PROGRAM P_Visu
VAR
	bFirstRun					: BOOL := TRUE;	
	
END_VAR

IF bFirstRun THEN
	bFirstRun := FALSE;
	FirstRun();
END_IF

JogButton();
SwitchButton();
SyncVariable();

METHOD FirstRun : BOOL
VAR_INPUT
END_VAR
GVL_VISU.stMachineConfig := P_Machine.MachineConfig;	
GVL_VISU.stCurMat := fbmat.Mat;
END_METHOD

METHOD JogButton : BOOL
VAR_INPUT
END_VAR
// JOG X
IF GVL_VISU.stMaintCmds.bJogXBw THEN
	GVL.fbMatAndToolHandling.JogX(TRUE);
ELSIF GVL_VISU.stMaintCmds.bJogXFw THEN
	GVL.fbMatAndToolHandling.JogX(FALSE);
ELSE
	GVL.fbMatAndToolHandling.JogXStop();
END_IF

// JOG Y
IF GVL_VISU.stMaintCmds.bJogYBw THEN
	GVL.fbMatAndToolHandling.JogY(TRUE);
ELSIF GVL_VISU.stMaintCmds.bJogYFw THEN
	GVL.fbMatAndToolHandling.JogY(FALSE);
ELSE
	GVL.fbMatAndToolHandling.JogYStop();
END_IF

// JOG Punch
IF GVL_VISU.stMaintCmds.bJogPunchBw THEN
	GVL.fbPunchEngine.Jog(FALSE, TRUE);
ELSIF GVL_VISU.stMaintCmds.bJogPunchFw THEN
	GVL.fbPunchEngine.Jog(TRUE, FALSE);
ELSE
	GVL.fbPunchEngine.JogStop();
END_IF

// JOG BELT
IF GVL_VISU.stMaintCmds.bJogOutletBelt THEN
	GVL.fbPunchEngine.OutletBeltJog(TRUE);
ELSE
	GVL.fbPunchEngine.OutletBeltJog(FALSE);
END_IF
END_METHOD

METHOD SwitchButton : BOOL
VAR_STAT
	stNullPunchCmds				: ST_PunchCmds;
	stNullMaintCmds				: ST_MaintCmds;
END_VAR
// PUNCH COMMANDS
IF MEMCMP(ADR(GVL_VISU.stPunchCmds), ADR(stNullPunchCmds), SIZEOF(ST_PunchCmds)) <> 0 THEN
	IF GVL_VISU.stPunchCmds.bLoad THEN
		P_Machine.LoadMat(GVL_VISU.stCurMat);		
		P_Machine.LoadJob(GVL_VISU.stPunchJob);	
	END_IF
	
	IF GVL_VISU.stPunchCmds.bStart THEN	
		P_Machine.LoadMat(GVL_VISU.stCurMat);	
		P_Machine.Start(GVL_VISU.stPunchJob);	
	END_IF
	
	IF GVL_VISU.stPunchCmds.bStop THEN
		P_Machine.Stop();	
	END_IF
	
	IF GVL_VISU.stPunchCmds.bResume THEN
		P_Machine.Resume();	
	END_IF
	
	IF GVL_VISU.stPunchCmds.bHalt THEN
		P_Machine.ClearJob();
		P_Machine.Halt();	
	END_IF	
		
	IF GVL_VISU.stPunchCmds.bLoadLeft THEN
		P_Machine.Maint(TRUE, TRUE, FALSE);	
	END_IF	
	
	IF GVL_VISU.stPunchCmds.bLoadRight THEN
		P_Machine.Maint(TRUE, TRUE, TRUE);	
	END_IF	
	
	IF GVL_VISU.stPunchCmds.bLoadStop THEN
		P_Machine.Halt();	
	END_IF	
	
	IF GVL_VISU.stPunchCmds.bUnlock THEN
		IF fbSafetyLock.Locked THEN
			GVL.fbSafetyLock.Unlock();
		ELSE
			GVL.fbSafetyLock.Lock();
		END_IF
	END_IF		
	
	IF GVL_VISU.stPunchCmds.bMoveTDC THEN
		GVL.fbPunchEngine.MoveTDC();	
	END_IF	
	
	IF GVL_VISU.stPunchCmds.bOutletBelt THEN
		GVL.fbPunchEngine.OutletBeltOnce();	
	END_IF	
		
	IF GVL_VISU.stPunchCmds.bOverride THEN
		P_Machine.Override := GVL_VISU.stPunchParam.fOverride;
	END_IF	
END_IF

// RESET PUNCH COMMANDS
GVL_VISU.stPunchCmds.bLoad := FALSE;
GVL_VISU.stPunchCmds.bStart := FALSE;
GVL_VISU.stPunchCmds.bStop := FALSE;
GVL_VISU.stPunchCmds.bResume := FALSE;
GVL_VISU.stPunchCmds.bHalt := FALSE;
GVL_VISU.stPunchCmds.bLoadLeft := FALSE;
GVL_VISU.stPunchCmds.bLoadRight := FALSE;
GVL_VISU.stPunchCmds.bMoveTDC := FALSE;
GVL_VISU.stPunchCmds.bOutletBelt := FALSE;
GVL_VISU.stPunchCmds.bOverride := FALSE;
GVL_VISU.stPunchCmds.bUnlock := FALSE;
GVL_VISU.stPunchCmds.bLoadStop := FALSE;

// MAINT COMMANDS
IF MEMCMP(ADR(GVL_VISU.stMaintCmds), ADR(stNullMaintCmds), SIZEOF(ST_MaintCmds)) <> 0 THEN	
	IF GVL_VISU.stMaintCmds.bLoadConfig THEN
		P_Machine.LoadConfig(GVL_VISU.stMachineConfig);
	END_IF
	
	IF GVL_VISU.stMaintCmds.bChangeTool THEN
		GVL.fbMatAndToolHandling.ChangeTool(GVL_VISU.stMaintParam.nChangeTool);
	END_IF
	
	IF GVL_VISU.stMaintCmds.bMoveXYMaint THEN
		P_Machine.Maint(TRUE, TRUE, FALSE);	
	END_IF
	
	IF GVL_VISU.stMaintCmds.bMoveXYMaintAlt THEN
		P_Machine.Maint(TRUE, TRUE, TRUE);	
	END_IF
	
	IF GVL_VISU.stMaintCmds.bReset THEN
		P_Machine.Reset();	
	END_IF	
	
	IF GVL_VISU.stMaintCmds.bMovePunchTDC THEN
		GVL.fbPunchEngine.MoveTDC();	
	END_IF	
	
	IF GVL_VISU.stMaintCmds.bSetZero THEN
		GVL.fbPunchEngine.SetZeroOffset();	
	END_IF	
	
END_IF

// RESET MAINT COMMANDS
GVL_VISU.stMaintCmds.bLoadConfig := FALSE;
GVL_VISU.stMaintCmds.bChangeTool := FALSE;
GVL_VISU.stMaintCmds.bMoveXYMaint := FALSE;
GVL_VISU.stMaintCmds.bMoveXYMaintAlt := FALSE;
GVL_VISU.stMaintCmds.bReset := FALSE;
GVL_VISU.stMaintCmds.bMovePunchTDC := FALSE; 
GVL_VISU.stMaintCmds.bSetZero := FALSE;
END_METHOD

METHOD SyncVariable : BOOL
VAR_INPUT
END_VAR
// VISU TO PLC
stPunchInfo.sCleartext 				:= P_Machine.seqOpMode.ClearText;
stPunchInfo.nCurMat 				:= P_Machine.CurMat + 1;
stPunchInfo.nCurPunch 				:= P_Machine.CurPunch + 1;
stPunchInfo.nCurRun 				:= P_Machine.CurRun + 1;
stPunchInfo.nMaxPunches 			:= P_Machine.MaxPunch + 1;
stPunchInfo.nCountRemainHolesOfJob 	:= P_Machine.CountRemainHolesOfJob + 1;
stPunchInfo.nCountAllHolesOfJob 	:= P_Machine.CountAllHolesOfJob + 1;
stPunchInfo.nRemainTimeOfJob 		:= P_Machine.RemainTimeOfJob;
stPunchInfo.stCoordinate 			:= P_Machine.stCoordinate;
stPunchInfo.bPunching 				:= P_Machine.Punching;
stPunchInfo.bResumeAllowed 			:= P_Machine.ResumeAllowed;
stPunchInfo.eJobState 				:= P_Machine.JobState;
stPunchInfo.fOverride 				:= P_Machine.Override;
stPunchInfo.fPunchspeed				:= fbPunchEngine.fbPunchAxis.Velocity;
stPunchInfo.bLocked					:= fbSafetyLock.Locked;

// X - Axis
stMaintInfo.bXHomed					:= fbMatAndToolHandling.fbAxisX.Homed;
stMaintInfo.bXError					:= fbMatAndToolHandling.fbAxisX.Error;
stMaintInfo.bXMoving				:= fbMatAndToolHandling.fbAxisX.Moving;
stMaintInfo.fXPosition				:= fbMatAndToolHandling.fbAxisX.ActPos;
stMaintInfo.fXTemp					:= fbMatAndToolHandling.fbAxisX.AmplifierTemp;
stMaintInfo.fXMotorTemp				:= fbMatAndToolHandling.fbAxisX.MotorTemp;
                            		   
// Y - Axis                 		   
stMaintInfo.bYHomed					:= fbMatAndToolHandling.fbAxisY.Homed;        
stMaintInfo.bYError					:= fbMatAndToolHandling.fbAxisY.Error;        
stMaintInfo.bYMoving				:= fbMatAndToolHandling.fbAxisY.Moving;       
stMaintInfo.fYPosition				:= fbMatAndToolHandling.fbAxisY.ActPos;       
stMaintInfo.fYTemp					:= fbMatAndToolHandling.fbAxisY.AmplifierTemp;
stMaintInfo.fYMotorTemp				:= fbMatAndToolHandling.fbAxisY.MotorTemp;    
                            		   
// Punch - Axis             		   
stMaintInfo.bPunchHomed				:= fbPunchEngine.fbPunchAxis.Homed;        
stMaintInfo.bPunchError				:= fbPunchEngine.fbPunchAxis.Error;        
stMaintInfo.bPunchMoving			:= fbPunchEngine.fbPunchAxis.Moving;       
stMaintInfo.fPunchPosition			:= fbPunchEngine.fbPunchAxis.ActModuloPos;       
stMaintInfo.fPunchTemp				:= fbPunchEngine.fbPunchAxis.AmplifierTemp;
stMaintInfo.fPunchMotorTemp			:= fbPunchEngine.fbPunchAxis.MotorTemp;   
 
// ToolChanger              		   
stMaintInfo.bToolError				:= fbMatAndToolHandling.fbToolSelector.State = E_ComponentState.eComponentState_error;
stMaintInfo.bToolChanged			:= fbMatAndToolHandling.ToolChanged;
stMaintInfo.nToolSelect				:= fbMatAndToolHandling.CurTool;
                            		   
// Machine                  		   
stMaintInfo.bSequenceError			:= P_Machine.seqOpMode.State = E_SequenceState.eSequenceState_error;
stMaintInfo.bSafetyOk				:= fbSafety.SafetyOk;
stMaintInfo.bEmergency				:= NOT fbSafety.bNotHaltOk;
stMaintInfo.nPunchCount				:= fbPunchEngine.PunchCount;                         		  
stMaintInfo.nStep					:= P_Machine.seqOpMode.Step;
stMaintInfo.nSequence				:= P_Machine.seqOpMode.SequenceId;
//stMaintInfo.bSafetyDoor				:= ;

// PLC TO VISU
P_Machine.CheckPosBeforeRun 		:= GVL_VISU.stPunchParam.bCheckPosBeforeRun;
END_METHOD

END_PROGRAM

(* stored: Version 1.1.0.1, ProductVersion 3.1.4022.12
   POU P_Visu: Id {fb0c63ef-be68-4ef0-98bb-ce4e496ecbe5}, SpecialFunc None
   Method FirstRun: Id {97d5756f-7d6c-467d-b24f-dc88368db921}
   Method JogButton: Id {4cba26b3-b30f-41c0-82fe-d8bffd0df9f6}
   Method SwitchButton: Id {79e15511-0af6-49f6-a7f8-55ac30540241}
   Method SyncVariable: Id {9e9d4bdf-b355-4f61-a9f5-0348c65df512} *)
